(* PLC project TC3_TE1400_GeneratedModule_Gewerk3_Simulinkmodell_2017_10_09_Twincat_FB, Beckhoff Automation GmbH & Co. KG TwinCAT 3 Function - TE1400 1.2.1229 *)
(* stored: companyURL www.beckhoff.com, creationDateTime 2017-10-10T13:37:05 *)

TYPE E_TcMatSimDataAreaType : (NotSpecified := 0, Standard, InputSrc, InputDst, OutputSrc, OutputDst, InternalDa, MArea, RetainDa);
END_TYPE

TYPE ST_TcMatSimObjectDataAreaInfo : STRUCT
  pPlcVar : PVOID;
  pModuleProcImg : PVOID;
  nSize : UDINT;
  nDataAreaId : UDINT;
  eDataAreaType : E_TcMatSimDataAreaType;
END_STRUCT;
END_TYPE

{attribute 'pack_mode' := '4'}
TYPE ST_Gewerk3_Simulinkmodell_2017_10_09_Twincat_InitData : STRUCT
  Header : TComInitDataHdr;
  CallByHdr : TComInitDataElmHdr;
  CallBy : TctModuleCallByType;
  ExecutionSequenceHdr : TComInitDataElmHdr;
  ExecutionSequence : TctModuleExecutionSequenceType;
  StepSizeHdr : TComInitDataElmHdr;
  StepSize : TctStepSizeType;
  ExecuteModelCodeHdr : TComInitDataElmHdr;
  ExecuteModelCode : BOOL;
  ModelParametersHdr : TComInitDataElmHdr;
  ModelParameters : P_Gewerk3_Simulinkmodell_2017_T;
  ContextInfoArr_0_TaskOidHdr : TComInitDataElmHdr;
  ContextInfoArr_0_TaskOid : OTCID;
  ContextInfoArr_0_TaskPriorityHdr : TComInitDataElmHdr;
  ContextInfoArr_0_TaskPriority : UDINT;
  ContextInfoArr_0_TaskCycleTimeNsHdr : TComInitDataElmHdr;
  ContextInfoArr_0_TaskCycleTimeNs : UDINT;
  ContextInfoArr_0_TaskPortHdr : TComInitDataElmHdr;
  ContextInfoArr_0_TaskPort : UINT;
  ContextInfoArr_0_TaskSortOrderHdr : TComInitDataElmHdr;
  ContextInfoArr_0_TaskSortOrder : UDINT;
END_STRUCT;
END_TYPE

TYPE ST_Gewerk3_Simulinkmodell_2017_10_09_Twincat_Input : STRUCT
  UDP : matrix_56_real_T;
  ProcessedData : matrix_15_real_T;
END_STRUCT;
END_TYPE

TYPE ST_Gewerk3_Simulinkmodell_2017_10_09_Twincat_Output : STRUCT
  cameradata : matrix_3_real_T;
  firstcameradatareceived : LREAL;
  cameradatavalid : LREAL;
  actualposition : matrix_3_real_T;
  L_theta : LREAL;
  L_x : LREAL;
  L_y : LREAL;
  v_x : LREAL;
  v_y : LREAL;
  v_theta : LREAL;
END_STRUCT;
END_TYPE

FUNCTION_BLOCK FB_TcMatSimObject
  VAR_INPUT
    bWriteFbInputValues : BOOL := TRUE;  (* set this flag to write FB input values to the TcComObject's input DataAreas. This will overwrite the mapped input values before module execution. Set to FALSE to read the mapped input values from the TcComObject to the FB. *)
  END_VAR
  VAR
    pDataAreas : POINTER TO ST_TcMatSimObjectDataAreaInfo;  (* process image src and dst pointers and sizes *)
    nDataAreas : UDINT;
    ipObjSrv : ITComObjectServer;  (* global interface pointers *)
    ipTcComObj : ITComObject;  (* object interface pointers *)
    ipTcCyclic : ITcCyclic;
    ipTcPostCyclic : ITcPostCyclic;
    ipTcAdi : ITcADI;
    ipTask : ITcTask;  (* task interface pointers *)
    pInitData : POINTER TO TComInitDataHdr;  (* initial parameters *)
    hResult : HRESULT;  (* hResult of interface calls (0 if no error) *)
    moduleClsId : CLSID;  (* module class ID *)
    assignedClsId : CLSID;  (* expected/desired module class ID *)
    bClassIdVerified : BOOL;
    bDynInstance : BOOL;  (* flag indicating whether the module instance was created dynamically *)
    eInitialObjState : TCOM_STATE := TCOM_STATE.TCOM_STATE_INIT;  (* the object state at the time FB_init was called, FB_exit will try to switch to this state (only if this means to shift down) *)
  END_VAR

            
          

{attribute 'object_name' := 'ReleaseTcComInterface'}
METHOD ReleaseTcComInterface : HRESULT
  VAR
    nStateChangeCnt : DINT := 0;
  END_VAR
                  
IF (ipTcComObj<>0) THEN
  WHILE (State>eInitialObjState AND nStateChangeCnt<1000) DO
    State := eInitialObjState;
    nStateChangeCnt := nStateChangeCnt+1;
  END_WHILE
  ReleaseObjInterfaces();
  IF (bDynInstance) THEN
    ReleaseTcComInterface := TC3_MODULE.FW_ObjMgr_DeleteInstance(ADR(ipTcComObj));
  ELSE
    ipTcComObj.TcRelease();
  END_IF
  ipTcComObj := 0;
END_IF
                  
                
END_METHOD

{attribute 'object_name' := 'ReleaseObjInterfaces'}
METHOD ReleaseObjInterfaces : HRESULT
                  
// release interface pointers
IF (ipTcCyclic<>0) THEN
  ipTcCyclic.TcRelease();
  ipTcCyclic := 0;
END_IF
IF (ipTcPostCyclic<>0) THEN
  ipTcPostCyclic.TcRelease();
  ipTcPostCyclic := 0;
END_IF
IF (ipTcAdi<>0) THEN
  ipTcAdi.TcRelease();
  ipTcAdi := 0;
END_IF
                  
                
END_METHOD

{attribute 'object_name' := 'Internal_SetObjState'}
METHOD Internal_SetObjState
  VAR_INPUT
    hr : REFERENCE TO HRESULT;
    nextState : TCOM_STATE;
  END_VAR
                  
// verify class id
IF (SUCCEEDED(hr)) THEN
  hr := VerifyClassId();
END_IF

// switch object state
IF (SUCCEEDED(hr) AND nextState>=TCOM_STATE_INIT) THEN
  IF (ipTcComObj=0) THEN
    hr := Tc2_System.E_HRESULTAdsErr.NOINTERFACE;
  END_IF
  IF (ipObjSrv=0) THEN
    hr := Tc2_System.E_HRESULTAdsErr.NOINTERFACE;
  END_IF
  IF (SUCCEEDED(hr)) THEN
    hr := ipTcComObj.TcSetObjState(nextState,ipObjSrv,pInitData);
  END_IF
END_IF
                  
                
END_METHOD

{attribute 'object_name' := 'FB_init'}
METHOD FB_init : BOOL
  VAR_INPUT
    bInitRetains : BOOL;  (* init retain variables *)
    bInCopyCode : BOOL;  (* Online Change *)
    oid : OTCID;
  END_VAR
                  
FB_init := SUCCEEDED(Init(oid));
                  
                
END_METHOD

{attribute 'object_name' := 'GetObjPara'}
METHOD GetObjPara : HRESULT
  VAR_INPUT
    pid : PTCID;
    nData : UDINT;
    pData : PVOID;
  END_VAR
                  
IF (ipTcComObj=0) THEN
  GetObjPara := Tc2_System.E_HRESULTAdsErr.NOINTERFACE;
END_IF

IF (SUCCEEDED(GetObjPara)) THEN
  GetObjPara := ipTcComObj.TcGetObjPara(pid:=pid,nData,pData,0);
END_IF
                  
                
END_METHOD

{attribute 'object_name' := 'QueryObjInterface'}
METHOD QueryObjInterface
  VAR_INPUT
    hr : REFERENCE TO HRESULT;
    iid : REFERENCE TO IID;
    pipItf : POINTER TO ITcUnknown;
  END_VAR
  VAR CONSTANT
    pNull : PVOID := 0;
  END_VAR
                  
IF (SUCCEEDED(hr)) THEN
  IF (ipTcComObj=0) THEN
    hr := Tc2_System.E_HRESULTAdsErr.NOINTERFACE;
  ELSIF (pipItf^=ULINT_TO_DWORD(pNull)) THEN
    hr := ipTcComObj.TcQueryInterface(iid:= iid, pipItf:=pipItf);
  END_IF
END_IF
                  
                
END_METHOD

{attribute 'object_name' := 'SaveOnlineParametersForInit'}
METHOD SaveOnlineParametersForInit : HRESULT
  VAR
    idx : UINT;
    pInitElemHdr : POINTER TO TComInitDataElmHdr;
    pData : PVOID;
    nData : UDINT;
  END_VAR
  VAR CONSTANT
    nInitDataAlignment : UDINT := 4;
  END_VAR
                  IF (pInitData<>0) THEN
  pInitElemHdr := pInitData + SIZEOF(pInitData^);
  FOR idx:=1 TO pInitData^.uiElmCnt DO
    pData := pInitElemHdr + ULINT_TO_DWORD(SIZEOF(pInitElemHdr^));
    nData := pInitElemHdr^.cbData;
    SaveOnlineParametersForInit := GetObjPara(pInitElemHdr^.indexOffset,nData,pData);
    IF (FAILED(SaveOnlineParametersForInit)) THEN
      RETURN;
    END_IF
    pInitElemHdr := pData + (nInitDataAlignment*((nData + nInitDataAlignment - 1)/nInitDataAlignment));
  END_FOR
ELSE
	SaveOnlineParametersForInit := Tc2_System.E_HRESULTAdsErr.NOTINIT;
END_IF
                  
                
END_METHOD

{attribute 'object_name' := 'ResetHresult'}
METHOD ResetHresult
                  hResult := S_OK;
                
END_METHOD

{attribute 'object_name' := 'Execute'}
METHOD Execute : HRESULT
  VAR
    nDaIdx : UDINT;
    pCurDataArea : POINTER TO ST_TcMatSimObjectDataAreaInfo;
  END_VAR
                  
IF (SUCCEEDED(hResult)) THEN
  hResult := VerifyClassId();
END_IF

IF (SUCCEEDED(hResult) AND State<>TCOM_STATE_OP) THEN
  hResult := Tc2_System.E_HRESULTAdsErr.NOTREADY;
END_IF

// get image pointers
IF (SUCCEEDED(hResult)) THEN
  GetImagePtrs(hResult);
END_IF

// copy inputs
IF (pDataAreas<>0 AND bWriteFbInputValues) THEN
  FOR nDaIdx:=0 TO nDataAreas-1 DO
    IF (FAILED(hResult))THEN
      CONTINUE;
    END_IF
    pCurDataArea := pDataAreas + nDaIdx*SIZEOF(ST_TcMatSimObjectDataAreaInfo);
    IF ((pCurDataArea^.eDataAreaType <> E_TcMatSimDataAreaType.InputDst))THEN
      CONTINUE;
    END_IF
    IF (pCurDataArea^.pModuleProcImg<>0 AND pCurDataArea^.pPlcVar<>0) THEN
      MEMCPY(pCurDataArea^.pModuleProcImg,pCurDataArea^.pPlcVar,pCurDataArea^.nSize);
    ELSE
      hResult := Tc2_System.E_HRESULTAdsErr.NOINTERFACE;
    END_IF
  END_FOR
END_IF

// call cycle update
IF (SUCCEEDED(hResult)) THEN
  IF (ipTcCyclic<>0) THEN
    hResult := ipTcCyclic.CycleUpdate(ipTask:= ipTask, ipCaller:= 0, context:= 0);
  ELSE
    hResult := Tc2_System.E_HRESULTAdsErr.NOINTERFACE;
  END_IF
END_IF

// copy outputs
IF (pDataAreas<>0) THEN
  FOR nDaIdx:=0 TO nDataAreas-1 DO
    IF (FAILED(hResult))THEN
      CONTINUE;
    END_IF
    pCurDataArea := pDataAreas + nDaIdx*SIZEOF(ST_TcMatSimObjectDataAreaInfo);
    IF ((pCurDataArea^.eDataAreaType = E_TcMatSimDataAreaType.OutputSrc) OR NOT bWriteFbInputValues) THEN
      IF (pCurDataArea^.pModuleProcImg<>0 AND pCurDataArea^.pPlcVar<>0) THEN
        MEMCPY(pCurDataArea^.pPlcVar,pCurDataArea^.pModuleProcImg,pCurDataArea^.nSize);
      ELSE
        hResult := Tc2_System.E_HRESULTAdsErr.NOINTERFACE;
      END_IF
    END_IF
  END_FOR
END_IF


// call post cyclic update
IF (SUCCEEDED(hResult)) THEN
  IF (ipTcPostCyclic<>0) THEN
    hResult := ipTcPostCyclic.PostCyclicUpdate(ipTask:= 0, ipCaller:= 0, context:= 0);
  ELSE
    hResult := Tc2_System.E_HRESULTAdsErr.NOINTERFACE;
  END_IF
END_IF

ReleaseImagePtrs();

Execute := hResult;
                  
                
END_METHOD

{attribute 'object_name' := 'GetImagePtrs'}
METHOD GetImagePtrs
  VAR_INPUT
    hr : REFERENCE TO HRESULT;
  END_VAR
  VAR
    nDaIdx : UDINT;
    pCurDataArea : POINTER TO ST_TcMatSimObjectDataAreaInfo;
  END_VAR
                  
IF (ipTcAdi=0) THEN
  hr := Tc2_System.E_HRESULTAdsErr.NOINTERFACE;
END_IF
IF(State<>TCOM_STATE_OP)THEN
  hr := Tc2_System.E_HRESULTAdsErr.INVALIDSTATE;
END_IF


// get pointers to process images
IF (pDataAreas<>0) THEN
  FOR nDaIdx:=0 TO nDataAreas-1 DO
    pCurDataArea := pDataAreas + nDaIdx*SIZEOF(ST_TcMatSimObjectDataAreaInfo);
    IF (FAILED(hr))THEN
      CONTINUE;
    END_IF
    IF ((pCurDataArea^.eDataAreaType <> E_TcMatSimDataAreaType.InputDst) AND (pCurDataArea^.eDataAreaType <> E_TcMatSimDataAreaType.OutputSrc))THEN
      CONTINUE;
    END_IF
    IF (pCurDataArea^.pModuleProcImg=0 AND pCurDataArea^.nSize>0) THEN
      hr := ipTcAdi.GetImagePtr(size:= pCurDataArea^.nSize , offs:=0 , adi_x:=pCurDataArea^.nDataAreaId , ppData:=ADR(pCurDataArea^.pModuleProcImg));
    END_IF
  END_FOR
END_IF

IF (FAILED(hr)) THEN
  ReleaseImagePtrs();
END_IF
                  
                
END_METHOD

{attribute 'object_name' := 'VerifyClassId'}
METHOD VerifyClassId : HRESULT
  VAR
    emptyClsId : CLSID;
  END_VAR
                  memset(ADR(emptyClsId),0,SIZEOF(emptyClsId));
IF (bClassIdVerified) THEN
  // class ID was already verified
  VerifyClassId := Tc2_System.E_HRESULTAdsErr.HRESULT_ADS_NOERROR;
ELSIF (memcmp(ADR(assignedClsId),ADR(emptyClsId),SIZEOF(assignedClsId))=0) THEN
  // skip class ID verification if no assignedClsId specified
  VerifyClassId := Tc2_System.E_HRESULTAdsErr.HRESULT_ADS_NOERROR;
ELSE
  // verify class ID
  VerifyClassId := ReadModuleClassId();

  IF (SUCCEEDED(VerifyClassId)) THEN
    IF (memcmp(ADR(assignedClsId),ADR(moduleClsId),SIZEOF(assignedClsId))<>0) THEN
     VerifyClassId := Tc2_System.E_HRESULTAdsErr.INVALIDCLSID;
    END_IF
  END_IF
  bClassIdVerified := SUCCEEDED(VerifyClassId);
END_IF
                  
                
END_METHOD

{attribute 'object_name' := 'SetObjPara'}
METHOD SetObjPara : HRESULT
  VAR_INPUT
    pid : PTCID;
    nData : UDINT;
    pData : PVOID;
  END_VAR
                  
IF (ipTcComObj=0) THEN
  SetObjPara := Tc2_System.E_HRESULTAdsErr.NOINTERFACE;
END_IF

IF (SUCCEEDED(SetObjPara)) THEN
  SetObjPara := ipTcComObj.TcSetObjPara(pid:=pid,nData,pData,0);
END_IF
                  
                
END_METHOD

{attribute 'object_name' := 'QueryTcComInterface'}
METHOD QueryTcComInterface
  VAR_INPUT
    hr : REFERENCE TO HRESULT;
    oid : OTCID;
  END_VAR
                  
IF (ipObjSrv=0) THEN
  hr := Tc2_System.E_HRESULTAdsErr.NOINTERFACE;
END_IF

IF (SUCCEEDED(hr) AND ipTcComObj=0) THEN
  bDynInstance := FALSE;
  IF(oid>0) THEN
    // query interface of existing object
    hr := ipObjSrv.TcQueryObjectInterface(oid,IID_ITComObject,ADR(ipTcComObj));
  ELSE
    // create new instance and get the object interface
    hr := ipObjSrv.TcCreateInstance(assignedClsId,IID_ITComObject,ADR(ipTcComObj));
    IF (SUCCEEDED(hr)) THEN
      bDynInstance := TRUE;
      hr := ipTcComObj.TcSetObjectId(OTCID_CreateNewId);
    END_IF
  END_IF
  IF (SUCCEEDED(hr)) THEN
    eInitialObjState := State;
  END_IF
END_IF
                  
                
END_METHOD

{attribute 'object_name' := 'ReleaseImagePtrs'}
METHOD ReleaseImagePtrs : HRESULT
  VAR
    nDaIdx : UDINT;
    pCurDataArea : POINTER TO ST_TcMatSimObjectDataAreaInfo;
  END_VAR
                  
IF (ipTcAdi=0) THEN
  ReleaseImagePtrs := Tc2_System.E_HRESULTAdsErr.NOINTERFACE;
END_IF

IF (SUCCEEDED(ReleaseImagePtrs) AND pDataAreas<>0) THEN
  // release pointers to the simulink module process images
  FOR nDaIdx:=0 TO nDataAreas-1 DO
    pCurDataArea := pDataAreas + nDaIdx*SIZEOF(ST_TcMatSimObjectDataAreaInfo);

    IF (pCurDataArea^.pModuleProcImg<>0) THEN
      ipTcAdi.ReleaseImagePtr(pData:=pCurDataArea^.pModuleProcImg);
      pCurDataArea^.pModuleProcImg := 0;
    END_IF
  END_FOR
END_IF
                  
                
END_METHOD

{attribute 'object_name' := 'FB_exit'}
METHOD FB_exit : BOOL
  VAR_INPUT
    bInCopyCode : BOOL;  (* Online Change *)
  END_VAR
                  
IF (NOT bInCopyCode) THEN
  IF (ipObjSrv<>0) THEN
    ipObjSrv.TcRelease();
    ipObjSrv := 0;
  END_IF

  ReleaseTcComInterface();
END_IF
                  
                
END_METHOD

{attribute 'object_name' := 'InitObjName'}
METHOD InitObjName
  VAR_INPUT
    hr : REFERENCE TO HRESULT;
  END_VAR
  VAR
    objectName : STRING(255) := 'TempContr_PlcRtFbInstance';
    oid : OTCID;
  END_VAR
                  
IF (SUCCEEDED(hr)) THEN
  hr := ipTcComObj.TcGetObjectId(oid);
END_IF

IF (SUCCEEDED(hr) and bDynInstance) THEN
  objectName := TC2_STANDARD.CONCAT(objectName,'_');
  objectName := TC2_STANDARD.CONCAT(objectName,UDINT_TO_STRING(oid));
  hr := ipTcComObj.TcSetObjectName(ADR(objectName));
END_IF
                  
                
END_METHOD

{attribute 'object_name' := 'SetObjState'}
METHOD SetObjState : HRESULT
  VAR_INPUT
    finalState : TCOM_STATE;
  END_VAR
  VAR
    bShiftUp : BOOL;
    bShiftDown : BOOL;
    currentState : TCOM_STATE;
  END_VAR
                  
currentState := State;

bShiftUp := finalState>currentState;
bShiftDown := finalState<currentState;

// do not switch up on error
IF (FAILED(hresult)) THEN
  bShiftUp := FALSE;
END_IF
// reset existing error on switching down
IF (bShiftDown) THEN
  ResetHresult();
END_IF

// prepared state switch
CASE currentState OF
  TCOM_STATE_INIT:
    IF(bShiftUp) THEN
      QueryTcComInterface(hResult,0);
      Internal_SetObjState(hResult,TCOM_STATE.TCOM_STATE_PREOP);
      InitObjName(hResult);
    END_IF

  TCOM_STATE_PREOP:
    IF(bShiftUp) THEN
      Internal_SetObjState(hResult,TCOM_STATE.TCOM_STATE_SAFEOP);
      QueryObjInterfaces(hResult);
    ELSIF (bShiftDown) THEN
      Internal_SetObjState(hResult,TCOM_STATE.TCOM_STATE_INIT);
    END_IF

  TCOM_STATE_SAFEOP:
    IF(bShiftUp) THEN
      Internal_SetObjState(hResult,TCOM_STATE.TCOM_STATE_OP);
      QueryObjInterfaces(hResult);
    ELSIF (bShiftDown) THEN
      Internal_SetObjState(hResult,TCOM_STATE.TCOM_STATE_PREOP);
      ReleaseObjInterfaces();
    END_IF


  TCOM_STATE_OP:
    IF (bShiftDown) THEN
      Internal_SetObjState(hResult,TCOM_STATE.TCOM_STATE_SAFEOP);
    END_IF
END_CASE

SetObjState := hResult;
                  
                
END_METHOD

{attribute 'object_name' := 'QueryObjInterfaces'}
METHOD QueryObjInterfaces
  VAR_INPUT
    hr : REFERENCE TO HRESULT;
  END_VAR
                  
IF(State<TCOM_STATE_PREOP)THEN
  hr := Tc2_System.E_HRESULTAdsErr.INVALIDSTATE;
END_IF

//cyclic interface
QueryObjInterface(hr,IID_ITCCYCLIC,ADR(ipTcCyclic));
//post cyclic interface
QueryObjInterface(hr,IID_ITCPOSTCYCLIC,ADR(ipTcPostCyclic));
//adi interface
QueryObjInterface(hr,IID_ITcADI,ADR(ipTcAdi));
                  
                
END_METHOD

{attribute 'object_name' := 'Init'}
METHOD Init : HRESULT
  VAR_INPUT
    oid : OTCID;
  END_VAR
                  
// preinitialize variables
memset(ADR(moduleClsId),0,SIZEOF(moduleClsId));
bClassIdVerified := FALSE;
hResult := Tc2_System.E_HRESULTAdsErr.HRESULT_ADS_NOERROR;

// get object server
IF (ipObjSrv=0) THEN
  hResult := FW_ObjMgr_GetObjectServer(_AppInfo.ObjId,ADR(ipObjSrv));
END_IF

// try to get object interfaces
IF (SUCCEEDED(hresult)) THEN
  QueryTcComInterface(hResult,oid);
END_IF

// verify class id
IF (SUCCEEDED(hresult)) THEN
  hresult := VerifyClassId();
END_IF

// query interfaces, if the current state is higher than INIT
IF (SUCCEEDED(hresult) AND State>TCOM_STATE.TCOM_STATE_INIT) THEN
  QueryObjInterfaces(hResult);
END_IF

// return value
Init := hresult;
                  
                
END_METHOD

{attribute 'object_name' := 'ReadModuleClassId'}
METHOD ReadModuleClassId : HRESULT
  VAR
    emptyClsId : CLSID;
  END_VAR
                  memset(ADR(emptyClsId),0,SIZEOF(emptyClsId));
IF (memcmp(ADR(moduleClsId),ADR(emptyClsId),SIZEOF(moduleClsId))=0) THEN
  IF (ipTcComObj=0) THEN
    ReadModuleClassId := Tc2_System.E_HRESULTAdsErr.NOINTERFACE;
  END_IF

  //objectClsId := clsid;
  IF (SUCCEEDED(ReadModuleClassId)) THEN
    ReadModuleClassId := ipTcComObj.GetClassId(moduleClsId);
  END_IF
END_IF
                
END_METHOD

METHOD PUBLIC AssignClassId
VAR_INPUT
	clsId : CLSID;
END_VAR
                  assignedClsId := clsId;
bClassIdVerified := false;
                  
                
END_METHOD

PROPERTY Error : BOOL
GET
                    Error := FAILED(hResult);
                  
END_GET
END_PROPERTY

METHOD PUBLIC SetDataAreaInfo
VAR_INPUT
  pDataAreas: POINTER TO ST_TcMatSimObjectDataAreaInfo;
  nDataAreas: UDINT;
END_VAR
                  
THIS^.nDataAreas := nDataAreas;
THIS^.pDataAreas := pDataAreas;
                  
                
END_METHOD

METHOD PUBLIC SetInitDataInfo
VAR_INPUT
  pInitData : POINTER TO TComInitDataHdr;
END_VAR
                  this^.pInitData := pInitData;
                
END_METHOD

PROPERTY ClassId : CLSID
GET
                    hResult := ReadModuleClassId();
ClassId := moduleClsId;
                    
                  
END_GET
END_PROPERTY

PROPERTY State : TCOM_STATE
GET
  VAR
    hr : HRESULT := S_OK;
    eObjState : TCOM_STATE;
  END_VAR
                    
IF (ipTcComObj<>0) THEN
  hr := ipTcComObj.TcGetObjState(ADR(eObjState));
IF (FAILED(hr)) THEN
  eObjState := TCOM_STATE.TCOM_STATE_INIT;
END_IF
ELSE
  eObjState := TCOM_STATE.TCOM_STATE_INIT;
END_IF
State := eObjState;
                    
                  
END_GET
SET
                    SetObjState(State);
                  
END_SET
END_PROPERTY

PROPERTY ErrorCode : HRESULT
GET
                    ErrorCode := hResult;
                  
END_GET
END_PROPERTY
END_FUNCTION_BLOCK

{attribute 'TcDependOnClassFactory' := 'Gewerk3_Simulinkmodell_2017_10_09_Twincat'}
FUNCTION_BLOCK FB_Gewerk3_Simulinkmodell_2017_10_09_Twincat EXTENDS FB_TcMatSimObject
  VAR_INPUT
    stInput : ST_Gewerk3_Simulinkmodell_2017_10_09_Twincat_Input;
  END_VAR
  VAR_OUTPUT
    stOutput : ST_Gewerk3_Simulinkmodell_2017_10_09_Twincat_Output;
  END_VAR
  VAR
    stInitData : ST_Gewerk3_Simulinkmodell_2017_10_09_Twincat_InitData;
    arrDataAreas : ARRAY[1..2] OF ST_TcMatSimObjectDataAreaInfo;
    bParametersVerified : BOOL;
  END_VAR

            
          

{attribute 'object_name' := 'Internal_SetObjState'}
METHOD Internal_SetObjState
  VAR_INPUT
    hr : REFERENCE TO HRESULT;
    nextState : TCOM_STATE;
  END_VAR
                  
// update pointer to InitData structure
SetInitDataInfo(ADR(stInitData));
// call base method
SUPER^.Internal_SetObjState(hr,nextState);
                  
                
END_METHOD

{attribute 'object_name' := 'SaveOnlineParametersForInit'}
METHOD SaveOnlineParametersForInit : HRESULT
  VAR
    idx : UINT;
    pInitElemHdr : POINTER TO TComInitDataElmHdr;
    pData : PVOID;
    nData : UDINT;
  END_VAR
  VAR CONSTANT
    nInitDataAlignment : UDINT := 4;
  END_VAR
                  
// update pointer to InitData structure
SetInitDataInfo(ADR(stInitData));
// call base method
SaveOnlineParametersForInit := SUPER^.SaveOnlineParametersForInit();
                  
                
END_METHOD

METHOD FB_init : BOOL
  VAR_INPUT
    bInitRetains : BOOL;  (* if TRUE, the retain variables are initialized (warm start / cold start) *)
    bInCopyCode : BOOL;  (* if TRUE, the instance afterwards gets moved into the copy code (online change) *)
    oid : OTCID;
  END_VAR
  VAR
    clsId : CLSID;
  END_VAR
                  
// initialize flags
bParametersVerified := false;
                    
// set module class id for compatibility check
clsId.Data1 := 16#6eb7a745;
clsId.Data2 := 16#175e;
clsId.Data3 := 16#42c9;
clsId.Data4[0] := 16#95;
clsId.Data4[1] := 16#b6;
clsId.Data4[2] := 16#2c;
clsId.Data4[3] := 16#25;
clsId.Data4[4] := 16#4f;
clsId.Data4[5] := 16#cf;
clsId.Data4[6] := 16#93;
clsId.Data4[7] := 16#48;

AssignClassId(clsId);
                    
// initialize InitData structure with default values              
stInitData.CallByHdr.indexGroup := 0;
stInitData.CallByHdr.indexOffset := 16#00000000;
stInitData.CallByHdr.cbData := SIZEOF(stInitData.CallBy);
stInitData.CallBy := TctModuleCallByType.CyclicTask;
stInitData.ExecutionSequenceHdr.indexGroup := 0;
stInitData.ExecutionSequenceHdr.indexOffset := 16#00000001;
stInitData.ExecutionSequenceHdr.cbData := SIZEOF(stInitData.ExecutionSequence);
stInitData.ExecutionSequence := TctModuleExecutionSequenceType.StateUpdateAfterOutputMapping;
stInitData.StepSizeHdr.indexGroup := 0;
stInitData.StepSizeHdr.indexOffset := 16#00000002;
stInitData.StepSizeHdr.cbData := SIZEOF(stInitData.StepSize);
stInitData.StepSize := TctStepSizeType.RequireMatchingTaskCycleTime;
stInitData.ExecuteModelCodeHdr.indexGroup := 0;
stInitData.ExecuteModelCodeHdr.indexOffset := 16#00000007;
stInitData.ExecuteModelCodeHdr.cbData := SIZEOF(stInitData.ExecuteModelCode);
stInitData.ExecuteModelCode := 1;
stInitData.ModelParametersHdr.indexGroup := 0;
stInitData.ModelParametersHdr.indexOffset := 16#83000000;
stInitData.ModelParametersHdr.cbData := SIZEOF(stInitData.ModelParameters);
stInitData.ModelParameters.K_1 := 12;
stInitData.ModelParameters.K_2 := 0.2;
stInitData.ModelParameters.L_konst := 10;
stInitData.ModelParameters.N := 12;
stInitData.ModelParameters.T_R := 0.03;
stInitData.ModelParameters.T_SP := 0.25;
stInitData.ModelParameters.accuracy_R := 1;
stInitData.ModelParameters.accuracy_Theta := 0.0174532925199433;
stInitData.ModelParameters.b_L_theta := 0.015;
stInitData.ModelParameters.b_L_x := 1.5;
stInitData.ModelParameters.b_L_y := 1.5;
stInitData.ModelParameters.m_L_theta := 0.01470360331117452;
stInitData.ModelParameters.m_L_x := 0.01903270296627266;
stInitData.ModelParameters.m_L_y := 0.01903270296627266;
stInitData.ModelParameters.omega_max := 2;
stInitData.ModelParameters.std_jitter := 0.011;
stInitData.ModelParameters.t_cam := 0.15;
stInitData.ModelParameters.t_cycle := 0.005;
stInitData.ModelParameters.v_max := 500;
stInitData.ModelParameters.var_cam_theta := 9e-06;
stInitData.ModelParameters.var_cam_x := 0.09;
stInitData.ModelParameters.var_cam_y := 0.09;
stInitData.ModelParameters.CompareToConstant_const := 1;
stInitData.ModelParameters.CompareToConstant1_const := 0;
stInitData.ModelParameters.CompareToConstant2_const := -1;
stInitData.ModelParameters.CompareToConstant3_const := 0;
stInitData.ModelParameters.CompareToConstant4_const := 0;
stInitData.ModelParameters.CompareToConstant_const_a := 1;
stInitData.ModelParameters.CompareToConstant1_const_f := 0;
stInitData.ModelParameters.CompareToConstant2_const_a := -1;
stInitData.ModelParameters.CompareToConstant3_const_c := 0;
stInitData.ModelParameters.CompareToConstant4_const_n := 0;
stInitData.ModelParameters.CompareToConstant_const_az := 1;
stInitData.ModelParameters.CompareToConstant1_const_p := 0;
stInitData.ModelParameters.CompareToConstant2_const_g := -1;
stInitData.ModelParameters.CompareToConstant3_const_n := 0;
stInitData.ModelParameters.CompareToConstant4_const_c := 0;
stInitData.ModelParameters.SRFlipFlop_initial_condition := 0;
stInitData.ModelParameters.SRFlipFlop1_initial_condition := 0;
stInitData.ModelParameters.driveforward_initial_condition := 0;
stInitData.ModelParameters.stationreached_initial_conditio := 0;
stInitData.ModelParameters.partavailable_initial_condition := 0;
stInitData.ModelParameters.grabberinprocess_initial_condit := 0;
stInitData.ModelParameters.opengrabber_initial_condition := 0;
stInitData.ModelParameters.readRFID_initial_condition := 0;
stInitData.ModelParameters.drivebackward_initial_condition := 0;
stInitData.ModelParameters.deactivatecontroller_initial_co := 0;
stInitData.ModelParameters.SRFlipFlop_initial_condition_f := 0;
stInitData.ModelParameters.startingpositionreached_initial := 0;
stInitData.ModelParameters.closegrabber_initial_condition := 0;
stInitData.ModelParameters.DetectRisePositive1_vinit := 0;
stInitData.ModelParameters.DetectRisePositive6_vinit := 0;
stInitData.ModelParameters.DetectRisePositive3_vinit := 0;
stInitData.ModelParameters.DetectRisePositive_vinit := 0;
stInitData.ModelParameters.DetectRisePositive_vinit_k := 0;
stInitData.ModelParameters.DetectRisePositive_vinit_p := 0;
stInitData.ModelParameters.DetectRisePositive_vinit_e := 0;
stInitData.ModelParameters.Gain2_Gain := 0.1591549430918953;
stInitData.ModelParameters.Gain2_Gain_f := 0.1591549430918953;
stInitData.ModelParameters.Constant_Value := 0;
stInitData.ModelParameters.Constant_Value_e := 0;
stInitData.ModelParameters.Constant_Value_o := 0;
stInitData.ModelParameters.Constant5_Value := 0;
stInitData.ModelParameters.Constant2_Value := 3.141592653589793;
stInitData.ModelParameters.Constant3_Value := 6.283185307179586;
stInitData.ModelParameters.Constant1_Value := 3.141592653589793;
stInitData.ModelParameters.Constant5_Value_h[0] := -150;
stInitData.ModelParameters.Constant5_Value_h[1] := 0;
stInitData.ModelParameters.Constant5_Value_h[2] := 0;
stInitData.ModelParameters.Constant_Value_m := 1;
stInitData.ModelParameters.Memory1_X0 := 0;
stInitData.ModelParameters.Switch2_Threshold := 0;
stInitData.ModelParameters.Constant2_Value_c := 3.141592653589793;
stInitData.ModelParameters.Constant3_Value_h := 6.283185307179586;
stInitData.ModelParameters.Constant1_Value_o := 3.141592653589793;
stInitData.ModelParameters.t_cycle_Delay := 0.5;
stInitData.ModelParameters.t_cycle_InitOutput := 0;
stInitData.ModelParameters.Constant_Value_l := 0;
stInitData.ModelParameters.Constant_Value_j := 0;
stInitData.ModelParameters.t_cycle_InitOutput_e := 0;
stInitData.ModelParameters.t_cycle_InitOutput_n := 0;
stInitData.ModelParameters.t_cycle_InitOutput_g := 0;
stInitData.ModelParameters.t_cycle_InitOutput_b := 0;
stInitData.ModelParameters.t_cycle_Delay_b := 0.5;
stInitData.ModelParameters.t_cycle_InitOutput_n4 := 0;
stInitData.ModelParameters.t_cycle_InitOutput_m := 0;
stInitData.ModelParameters.t_cycle_InitOutput_p := 0;
stInitData.ModelParameters.t_cycle_Delay_a := 0.5;
stInitData.ModelParameters.t_cycle_InitOutput_f := 0;
stInitData.ModelParameters.t_cycle_InitOutput_i := 0;
stInitData.ModelParameters.t_cycle_InitOutput_k := 0;
stInitData.ModelParameters.t_cycle_Delay_o := 2;
stInitData.ModelParameters.t_cycle_InitOutput_a := 0;
stInitData.ModelParameters.t_cycle_InitOutput_h := 0;
stInitData.ModelParameters.Constant1_Value_m[0] := 150;
stInitData.ModelParameters.Constant1_Value_m[1] := 0;
stInitData.ModelParameters.Constant1_Value_m[2] := 0;
stInitData.ModelParameters.Constant4_Value[0] := 0;
stInitData.ModelParameters.Constant4_Value[1] := 0;
stInitData.ModelParameters.Constant4_Value[2] := 0;
stInitData.ModelParameters.u5sek_Delay := 0.5;
stInitData.ModelParameters.u5sek_InitOutput := 0;
stInitData.ModelParameters.Constant1_Value_oa := 3.141592653589793;
stInitData.ModelParameters.Constant2_Value_h := 6.283185307179586;
stInitData.ModelParameters.Constant3_Value_k := 3.141592653589793;
stInitData.ModelParameters.Constant1_Value_f := 3.141592653589793;
stInitData.ModelParameters.Constant2_Value_e := 6.283185307179586;
stInitData.ModelParameters.Constant3_Value_c := 3.141592653589793;
stInitData.ModelParameters.Constant2_Value_i := 6.283185307179586;
stInitData.ModelParameters.UnitDelay2_InitialCondition := 0;
stInitData.ModelParameters.UnitDelay2_InitialCondition_c := 0;
stInitData.ModelParameters.cameradeadtime_InitOutput := 0;
stInitData.ModelParameters.Constant2_Value_k[0] := 0;
stInitData.ModelParameters.Constant2_Value_k[1] := 0;
stInitData.ModelParameters.Constant2_Value_k[2] := 0;
stInitData.ModelParameters.Constant2_Value_a := 6.283185307179586;
stInitData.ModelParameters.Constant1_Value_i := 3.141592653589793;
stInitData.ModelParameters.Constant2_Value_e3 := 6.283185307179586;
stInitData.ModelParameters.Constant3_Value_kp := 3.141592653589793;
stInitData.ModelParameters.Constant1_Value_n[0] := 0;
stInitData.ModelParameters.Constant1_Value_n[1] := 0;
stInitData.ModelParameters.Constant1_Value_n[2] := 0;
stInitData.ModelParameters.Constant_Value_f := 0;
stInitData.ModelParameters.Constant4_Value_d := 0;
stInitData.ModelParameters.cameradeadtime_InitOutput_a := 0;
stInitData.ModelParameters.Constant2_Value_d := 3.141592653589793;
stInitData.ModelParameters.Constant3_Value_m := 6.283185307179586;
stInitData.ModelParameters.Constant1_Value_mh := 3.141592653589793;
stInitData.ModelParameters.Constant_Value_g := 0;
stInitData.ModelParameters.cameradeadtime_InitOutput_b := 0;
stInitData.ModelParameters.Constant_Value_d := 0;
stInitData.ModelParameters.cameradeadtime_InitOutput_k := 0;
stInitData.ModelParameters.u8sek_Delay := 0.8;
stInitData.ModelParameters.u8sek_InitOutput := 0;
stInitData.ModelParameters.t_cycle_InitOutput_bp := 0;
stInitData.ModelParameters.Constant1_Value_g := 3.141592653589793;
stInitData.ModelParameters.Constant2_Value_f := 6.283185307179586;
stInitData.ModelParameters.Constant3_Value_e := 3.141592653589793;
stInitData.ModelParameters.UnitDelay2_InitialCondition_m := 0;
stInitData.ModelParameters.Constant1_Value_d := 3.141592653589793;
stInitData.ModelParameters.Constant2_Value_fr := 6.283185307179586;
stInitData.ModelParameters.Constant3_Value_cs := 3.141592653589793;
stInitData.ModelParameters.Constant_Value_oc := 0;
stInitData.ModelParameters.Constant1_Value_fq := 3.141592653589793;
stInitData.ModelParameters.Constant2_Value_ak := 6.283185307179586;
stInitData.ModelParameters.Constant3_Value_mf := 3.141592653589793;
stInitData.ModelParameters.Switch2_Threshold_o := 0;
stInitData.ModelParameters.Constant_Value_h := 0;
stInitData.ModelParameters.Switch2_Threshold_c := 0;
stInitData.ModelParameters.Constant_Value_ho := 0;
stInitData.ModelParameters.Switch2_Threshold_d := 0;
stInitData.ModelParameters.t_cycle_InitOutput_j := 0;
stInitData.ModelParameters.ManualSwitch_CurrentSetting := 0;
stInitData.ModelParameters.ManualSwitch_CurrentSetting_l := 0;
stInitData.ModelParameters.ManualSwitch_CurrentSetting_ly := 0;
stInitData.ModelParameters.UnitDelay_InitialCondition := 0;
stInitData.ModelParameters.ManualSwitch_CurrentSetting_d := 0;
stInitData.ModelParameters.Logic_table[0] := 0;
stInitData.ModelParameters.Logic_table[1] := 1;
stInitData.ModelParameters.Logic_table[2] := 0;
stInitData.ModelParameters.Logic_table[3] := 0;
stInitData.ModelParameters.Logic_table[4] := 1;
stInitData.ModelParameters.Logic_table[5] := 1;
stInitData.ModelParameters.Logic_table[6] := 0;
stInitData.ModelParameters.Logic_table[7] := 0;
stInitData.ModelParameters.Logic_table[8] := 1;
stInitData.ModelParameters.Logic_table[9] := 0;
stInitData.ModelParameters.Logic_table[10] := 1;
stInitData.ModelParameters.Logic_table[11] := 1;
stInitData.ModelParameters.Logic_table[12] := 0;
stInitData.ModelParameters.Logic_table[13] := 0;
stInitData.ModelParameters.Logic_table[14] := 0;
stInitData.ModelParameters.Logic_table[15] := 0;
stInitData.ModelParameters.Constant_Value_g4 := 0;
stInitData.ModelParameters.Logic_table_c[0] := 0;
stInitData.ModelParameters.Logic_table_c[1] := 1;
stInitData.ModelParameters.Logic_table_c[2] := 0;
stInitData.ModelParameters.Logic_table_c[3] := 0;
stInitData.ModelParameters.Logic_table_c[4] := 1;
stInitData.ModelParameters.Logic_table_c[5] := 1;
stInitData.ModelParameters.Logic_table_c[6] := 0;
stInitData.ModelParameters.Logic_table_c[7] := 0;
stInitData.ModelParameters.Logic_table_c[8] := 1;
stInitData.ModelParameters.Logic_table_c[9] := 0;
stInitData.ModelParameters.Logic_table_c[10] := 1;
stInitData.ModelParameters.Logic_table_c[11] := 1;
stInitData.ModelParameters.Logic_table_c[12] := 0;
stInitData.ModelParameters.Logic_table_c[13] := 0;
stInitData.ModelParameters.Logic_table_c[14] := 0;
stInitData.ModelParameters.Logic_table_c[15] := 0;
stInitData.ModelParameters.UnitDelay_InitialCondition_a := 0;
stInitData.ModelParameters.Logic_table_p[0] := 0;
stInitData.ModelParameters.Logic_table_p[1] := 1;
stInitData.ModelParameters.Logic_table_p[2] := 0;
stInitData.ModelParameters.Logic_table_p[3] := 0;
stInitData.ModelParameters.Logic_table_p[4] := 1;
stInitData.ModelParameters.Logic_table_p[5] := 1;
stInitData.ModelParameters.Logic_table_p[6] := 0;
stInitData.ModelParameters.Logic_table_p[7] := 0;
stInitData.ModelParameters.Logic_table_p[8] := 1;
stInitData.ModelParameters.Logic_table_p[9] := 0;
stInitData.ModelParameters.Logic_table_p[10] := 1;
stInitData.ModelParameters.Logic_table_p[11] := 1;
stInitData.ModelParameters.Logic_table_p[12] := 0;
stInitData.ModelParameters.Logic_table_p[13] := 0;
stInitData.ModelParameters.Logic_table_p[14] := 0;
stInitData.ModelParameters.Logic_table_p[15] := 0;
stInitData.ModelParameters.Logic_table_b[0] := 0;
stInitData.ModelParameters.Logic_table_b[1] := 1;
stInitData.ModelParameters.Logic_table_b[2] := 0;
stInitData.ModelParameters.Logic_table_b[3] := 0;
stInitData.ModelParameters.Logic_table_b[4] := 1;
stInitData.ModelParameters.Logic_table_b[5] := 1;
stInitData.ModelParameters.Logic_table_b[6] := 0;
stInitData.ModelParameters.Logic_table_b[7] := 0;
stInitData.ModelParameters.Logic_table_b[8] := 1;
stInitData.ModelParameters.Logic_table_b[9] := 0;
stInitData.ModelParameters.Logic_table_b[10] := 1;
stInitData.ModelParameters.Logic_table_b[11] := 1;
stInitData.ModelParameters.Logic_table_b[12] := 0;
stInitData.ModelParameters.Logic_table_b[13] := 0;
stInitData.ModelParameters.Logic_table_b[14] := 0;
stInitData.ModelParameters.Logic_table_b[15] := 0;
stInitData.ModelParameters.Logic_table_l[0] := 0;
stInitData.ModelParameters.Logic_table_l[1] := 1;
stInitData.ModelParameters.Logic_table_l[2] := 0;
stInitData.ModelParameters.Logic_table_l[3] := 0;
stInitData.ModelParameters.Logic_table_l[4] := 1;
stInitData.ModelParameters.Logic_table_l[5] := 1;
stInitData.ModelParameters.Logic_table_l[6] := 0;
stInitData.ModelParameters.Logic_table_l[7] := 0;
stInitData.ModelParameters.Logic_table_l[8] := 1;
stInitData.ModelParameters.Logic_table_l[9] := 0;
stInitData.ModelParameters.Logic_table_l[10] := 1;
stInitData.ModelParameters.Logic_table_l[11] := 1;
stInitData.ModelParameters.Logic_table_l[12] := 0;
stInitData.ModelParameters.Logic_table_l[13] := 0;
stInitData.ModelParameters.Logic_table_l[14] := 0;
stInitData.ModelParameters.Logic_table_l[15] := 0;
stInitData.ModelParameters.Logic_table_i[0] := 0;
stInitData.ModelParameters.Logic_table_i[1] := 1;
stInitData.ModelParameters.Logic_table_i[2] := 0;
stInitData.ModelParameters.Logic_table_i[3] := 0;
stInitData.ModelParameters.Logic_table_i[4] := 1;
stInitData.ModelParameters.Logic_table_i[5] := 1;
stInitData.ModelParameters.Logic_table_i[6] := 0;
stInitData.ModelParameters.Logic_table_i[7] := 0;
stInitData.ModelParameters.Logic_table_i[8] := 1;
stInitData.ModelParameters.Logic_table_i[9] := 0;
stInitData.ModelParameters.Logic_table_i[10] := 1;
stInitData.ModelParameters.Logic_table_i[11] := 1;
stInitData.ModelParameters.Logic_table_i[12] := 0;
stInitData.ModelParameters.Logic_table_i[13] := 0;
stInitData.ModelParameters.Logic_table_i[14] := 0;
stInitData.ModelParameters.Logic_table_i[15] := 0;
stInitData.ModelParameters.Logic_table_pn[0] := 0;
stInitData.ModelParameters.Logic_table_pn[1] := 1;
stInitData.ModelParameters.Logic_table_pn[2] := 0;
stInitData.ModelParameters.Logic_table_pn[3] := 0;
stInitData.ModelParameters.Logic_table_pn[4] := 1;
stInitData.ModelParameters.Logic_table_pn[5] := 1;
stInitData.ModelParameters.Logic_table_pn[6] := 0;
stInitData.ModelParameters.Logic_table_pn[7] := 0;
stInitData.ModelParameters.Logic_table_pn[8] := 1;
stInitData.ModelParameters.Logic_table_pn[9] := 0;
stInitData.ModelParameters.Logic_table_pn[10] := 1;
stInitData.ModelParameters.Logic_table_pn[11] := 1;
stInitData.ModelParameters.Logic_table_pn[12] := 0;
stInitData.ModelParameters.Logic_table_pn[13] := 0;
stInitData.ModelParameters.Logic_table_pn[14] := 0;
stInitData.ModelParameters.Logic_table_pn[15] := 0;
stInitData.ModelParameters.Logic_table_h[0] := 0;
stInitData.ModelParameters.Logic_table_h[1] := 1;
stInitData.ModelParameters.Logic_table_h[2] := 0;
stInitData.ModelParameters.Logic_table_h[3] := 0;
stInitData.ModelParameters.Logic_table_h[4] := 1;
stInitData.ModelParameters.Logic_table_h[5] := 1;
stInitData.ModelParameters.Logic_table_h[6] := 0;
stInitData.ModelParameters.Logic_table_h[7] := 0;
stInitData.ModelParameters.Logic_table_h[8] := 1;
stInitData.ModelParameters.Logic_table_h[9] := 0;
stInitData.ModelParameters.Logic_table_h[10] := 1;
stInitData.ModelParameters.Logic_table_h[11] := 1;
stInitData.ModelParameters.Logic_table_h[12] := 0;
stInitData.ModelParameters.Logic_table_h[13] := 0;
stInitData.ModelParameters.Logic_table_h[14] := 0;
stInitData.ModelParameters.Logic_table_h[15] := 0;
stInitData.ModelParameters.Logic_table_e[0] := 0;
stInitData.ModelParameters.Logic_table_e[1] := 1;
stInitData.ModelParameters.Logic_table_e[2] := 0;
stInitData.ModelParameters.Logic_table_e[3] := 0;
stInitData.ModelParameters.Logic_table_e[4] := 1;
stInitData.ModelParameters.Logic_table_e[5] := 1;
stInitData.ModelParameters.Logic_table_e[6] := 0;
stInitData.ModelParameters.Logic_table_e[7] := 0;
stInitData.ModelParameters.Logic_table_e[8] := 1;
stInitData.ModelParameters.Logic_table_e[9] := 0;
stInitData.ModelParameters.Logic_table_e[10] := 1;
stInitData.ModelParameters.Logic_table_e[11] := 1;
stInitData.ModelParameters.Logic_table_e[12] := 0;
stInitData.ModelParameters.Logic_table_e[13] := 0;
stInitData.ModelParameters.Logic_table_e[14] := 0;
stInitData.ModelParameters.Logic_table_e[15] := 0;
stInitData.ModelParameters.Logic_table_cl[0] := 0;
stInitData.ModelParameters.Logic_table_cl[1] := 1;
stInitData.ModelParameters.Logic_table_cl[2] := 0;
stInitData.ModelParameters.Logic_table_cl[3] := 0;
stInitData.ModelParameters.Logic_table_cl[4] := 1;
stInitData.ModelParameters.Logic_table_cl[5] := 1;
stInitData.ModelParameters.Logic_table_cl[6] := 0;
stInitData.ModelParameters.Logic_table_cl[7] := 0;
stInitData.ModelParameters.Logic_table_cl[8] := 1;
stInitData.ModelParameters.Logic_table_cl[9] := 0;
stInitData.ModelParameters.Logic_table_cl[10] := 1;
stInitData.ModelParameters.Logic_table_cl[11] := 1;
stInitData.ModelParameters.Logic_table_cl[12] := 0;
stInitData.ModelParameters.Logic_table_cl[13] := 0;
stInitData.ModelParameters.Logic_table_cl[14] := 0;
stInitData.ModelParameters.Logic_table_cl[15] := 0;
stInitData.ModelParameters.Constant_Value_ja := 0;
stInitData.ModelParameters.UnitDelay1_InitialCondition := 0;
stInitData.ModelParameters.Constant_Value_f0 := 0;
stInitData.ModelParameters.UnitDelay1_InitialCondition_k := 0;
stInitData.ModelParameters.Constant_Value_n := 0;
stInitData.ModelParameters.UnitDelay1_InitialCondition_i := 0;
stInitData.ModelParameters.UnitDelay2_InitialCondition_ca := 0;
stInitData.ModelParameters.Logic_table_le[0] := 0;
stInitData.ModelParameters.Logic_table_le[1] := 1;
stInitData.ModelParameters.Logic_table_le[2] := 0;
stInitData.ModelParameters.Logic_table_le[3] := 0;
stInitData.ModelParameters.Logic_table_le[4] := 1;
stInitData.ModelParameters.Logic_table_le[5] := 1;
stInitData.ModelParameters.Logic_table_le[6] := 0;
stInitData.ModelParameters.Logic_table_le[7] := 0;
stInitData.ModelParameters.Logic_table_le[8] := 1;
stInitData.ModelParameters.Logic_table_le[9] := 0;
stInitData.ModelParameters.Logic_table_le[10] := 1;
stInitData.ModelParameters.Logic_table_le[11] := 1;
stInitData.ModelParameters.Logic_table_le[12] := 0;
stInitData.ModelParameters.Logic_table_le[13] := 0;
stInitData.ModelParameters.Logic_table_le[14] := 0;
stInitData.ModelParameters.Logic_table_le[15] := 0;
stInitData.ModelParameters.Logic_table_o[0] := 0;
stInitData.ModelParameters.Logic_table_o[1] := 1;
stInitData.ModelParameters.Logic_table_o[2] := 0;
stInitData.ModelParameters.Logic_table_o[3] := 0;
stInitData.ModelParameters.Logic_table_o[4] := 1;
stInitData.ModelParameters.Logic_table_o[5] := 1;
stInitData.ModelParameters.Logic_table_o[6] := 0;
stInitData.ModelParameters.Logic_table_o[7] := 0;
stInitData.ModelParameters.Logic_table_o[8] := 1;
stInitData.ModelParameters.Logic_table_o[9] := 0;
stInitData.ModelParameters.Logic_table_o[10] := 1;
stInitData.ModelParameters.Logic_table_o[11] := 1;
stInitData.ModelParameters.Logic_table_o[12] := 0;
stInitData.ModelParameters.Logic_table_o[13] := 0;
stInitData.ModelParameters.Logic_table_o[14] := 0;
stInitData.ModelParameters.Logic_table_o[15] := 0;
stInitData.ModelParameters.UnitDelay1_InitialCondition_l := 0;
stInitData.ModelParameters.Constant_Value_fx := 0;
stInitData.ModelParameters.Constant_Value_hor := 0;
stInitData.ModelParameters.Logic_table_iw[0] := 0;
stInitData.ModelParameters.Logic_table_iw[1] := 1;
stInitData.ModelParameters.Logic_table_iw[2] := 0;
stInitData.ModelParameters.Logic_table_iw[3] := 0;
stInitData.ModelParameters.Logic_table_iw[4] := 1;
stInitData.ModelParameters.Logic_table_iw[5] := 1;
stInitData.ModelParameters.Logic_table_iw[6] := 0;
stInitData.ModelParameters.Logic_table_iw[7] := 0;
stInitData.ModelParameters.Logic_table_iw[8] := 1;
stInitData.ModelParameters.Logic_table_iw[9] := 0;
stInitData.ModelParameters.Logic_table_iw[10] := 1;
stInitData.ModelParameters.Logic_table_iw[11] := 1;
stInitData.ModelParameters.Logic_table_iw[12] := 0;
stInitData.ModelParameters.Logic_table_iw[13] := 0;
stInitData.ModelParameters.Logic_table_iw[14] := 0;
stInitData.ModelParameters.Logic_table_iw[15] := 0;
stInitData.ContextInfoArr_0_TaskOidHdr.indexGroup := 0;
stInitData.ContextInfoArr_0_TaskOidHdr.indexOffset := 16#03002060;
stInitData.ContextInfoArr_0_TaskOidHdr.cbData := SIZEOF(stInitData.ContextInfoArr_0_TaskOid);
stInitData.ContextInfoArr_0_TaskPriorityHdr.indexGroup := 0;
stInitData.ContextInfoArr_0_TaskPriorityHdr.indexOffset := 16#03002070;
stInitData.ContextInfoArr_0_TaskPriorityHdr.cbData := SIZEOF(stInitData.ContextInfoArr_0_TaskPriority);
stInitData.ContextInfoArr_0_TaskCycleTimeNsHdr.indexGroup := 0;
stInitData.ContextInfoArr_0_TaskCycleTimeNsHdr.indexOffset := 16#03002080;
stInitData.ContextInfoArr_0_TaskCycleTimeNsHdr.cbData := SIZEOF(stInitData.ContextInfoArr_0_TaskCycleTimeNs);
stInitData.ContextInfoArr_0_TaskPortHdr.indexGroup := 0;
stInitData.ContextInfoArr_0_TaskPortHdr.indexOffset := 16#03002090;
stInitData.ContextInfoArr_0_TaskPortHdr.cbData := SIZEOF(stInitData.ContextInfoArr_0_TaskPort);
stInitData.ContextInfoArr_0_TaskSortOrderHdr.indexGroup := 0;
stInitData.ContextInfoArr_0_TaskSortOrderHdr.indexOffset := 16#030020b0;
stInitData.ContextInfoArr_0_TaskSortOrderHdr.cbData := SIZEOF(stInitData.ContextInfoArr_0_TaskSortOrder);
stInitData.Header.cbData := SIZEOF(stInitData)-SIZEOF(stInitData.Header);
stInitData.Header.uiElmCnt := 10;


// set pointer to InitData structure
SetInitDataInfo(ADR(stInitData));

// set DataArea information
SetDataAreaInfo(ADR(arrDataAreas),2);
arrDataAreas[1].nDataAreaId := 0;
arrDataAreas[1].nSize := SIZEOF(stInput);
arrDataAreas[1].pPlcVar := ADR(stInput);
arrDataAreas[1].pModuleProcImg := 0;
arrDataAreas[1].eDataAreaType := E_TcMatSimDataAreaType.InputDst;
arrDataAreas[2].nDataAreaId := 1;
arrDataAreas[2].nSize := SIZEOF(stOutput);
arrDataAreas[2].pPlcVar := ADR(stOutput);
arrDataAreas[2].pModuleProcImg := 0;
arrDataAreas[2].eDataAreaType := E_TcMatSimDataAreaType.OutputSrc;


// initialize basic interface pointers and return
FB_init := SUCCEEDED(Init(oid));
                  
                
END_METHOD

METHOD Execute : HRESULT
                  
IF (SUCCEEDED(hResult)) THEN
  hResult := VerifyParameters();
END_IF

	// update DataArea information
SetDataAreaInfo(ADR(arrDataAreas),2);
	
	// call base method
Execute := SUPER^.Execute();
                  
                
END_METHOD

{attribute 'object_name' := 'VerifyParameters'}
METHOD VerifyParameters : HRESULT
  VAR
    moduleCallByParam : TctModuleCallByType;
  END_VAR
                  
IF (bParametersVerified) THEN
  VerifyParameters := Tc2_System.E_HRESULTAdsErr.HRESULT_ADS_NOERROR;
ELSE
  VerifyParameters := GetObjPara(stInitData.CallByHdr.indexOffset,SIZEOF(moduleCallByParam),ADR(moduleCallByParam));
  
  // check the "CallBy" parameter to be set to "Module"
  IF (SUCCEEDED(VerifyParameters) AND (moduleCallByParam <> TctModuleCallByType.Module)) THEN
      VerifyParameters := Tc2_System.E_HRESULTAdsErr.INVALIDPARM;
  END_IF
  
  // set the parameters verified flag
  bParametersVerified := SUCCEEDED(VerifyParameters);
END_IF
                  
                
END_METHOD

PROPERTY InitData : ST_Gewerk3_Simulinkmodell_2017_10_09_Twincat_InitData
GET
                    InitData := stInitData;
                  
END_GET
SET
                    stInitData := InitData;
                  
END_SET
END_PROPERTY
END_FUNCTION_BLOCK
